// TIA Portal V19 export
TYPE "LEXCHANGETRAY_typePlasticEm5_toRollerDeliver"
// stored: Access Published
   STRUCT
      feedback : "LEXCHANGETRAY_typePlasticEm5_toRollerFeedback";
      req : "LEXCHANGETRAY_typePlasticEm5_toRollerReq";
   END_STRUCT;
END_TYPE
